FUNCTION_BLOCK FB_Mover_1 EXTENDS FB_Mover
VAR_INPUT
END_VAR
VAR_OUTPUT
END_VAR
VAR
END_VAR

SUPER^();

METHOD M_MoveToPickPos : BOOL
VAR_INPUT
END_VAR
//If Mover1 then PickFromCassette; if Mover2  PickFromBuffer

//State := E_MoverTransitionState.Picking;


Sim_Time(IN := TRUE, PT := T#1S);

IF Sim_Time.Q THEN       //We assume in 1 seconds we go to Pick position; CassettePos for Mover1, BufferPos for Mover2
	Sim_Time(IN := FALSE);
	State := E_MoverFixedState.InPickedPos;
END_IF
END_METHOD

METHOD M_MoveToPlacePos : BOOL
VAR_INPUT
	Buffer_1_InUse : BOOL;
	Buffer_Pos : INT;
END_VAR
//If Mover1 then PlaceToCarrier; if Mover2  PlaceToBuffer
//State := E_MoverTransitionState.Placing;


Sim_Time(IN := TRUE, PT := T#1S);

IF Sim_Time.Q THEN   //We assume in 1 seconds we go to Pick position; BufferPos for Mover1, CarrierPos for Mover2
	Sim_Time(IN := FALSE);
	State := E_MoverFixedState.InPlacedPos;
END_IF
END_METHOD

END_FUNCTION_BLOCK

(* stored: Version 1.1.0.1, ProductVersion 3.1.4024.12
   POU FB_Mover_1: Id {91297915-e066-40a2-a7f5-28d2930e8691}, SpecialFunc None
   Method M_MoveToPickPos: Id {f64fc3ca-7148-49e5-9864-e4dee441f6e8}
   Method M_MoveToPlacePos: Id {2e459992-cfe1-4ff9-ad47-0e875ce65f90} *)
